{attribute 'qualified_only'}
VAR_GLOBAL CONSTANT
    C_MaxSyncUnits : UINT := 10;
	C_MAX_LOCAL_ERROR_MESSAGES : UINT := 3;	
END_VAR

(* stored: Version 1.1.0.1, ProductVersion 3.1.4024.9
   GVL TcoEthercat: Id {70ccb30f-a686-0e63-2d40-73db5f7a8607} *)
